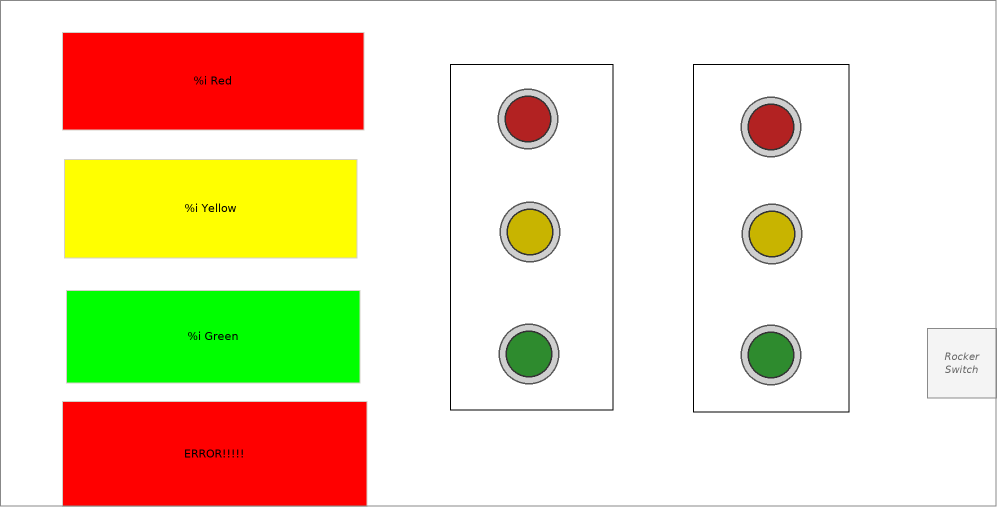
VISUALIZATION Visualization  // 997x507
    Rectangle (450,64 163x346)
    Lamp1 (494,319 70x70), variable: TrafficLight.bGreenLight, style: Lamp-Lamp1-Green
    Lamp1 (495,197 70x70), variable: TrafficLight.bYellowLight, style: Lamp-Lamp1-Yellow
    Lamp1 (493,84 70x70), variable: TrafficLight.bRedLight, style: Lamp-Lamp1-Red
    RockerSwitch (927,328 70x70), variable: TrafficLight.bTurnOnVis, behaviour: TOGGLE, style: Switch-RockerSwitch-Red
    Textfield (62,32 302x98), "%i Red", text variable: TrafficLight.iRedColor
        OnMouseDown: write the text variable via Default
    Textfield (64,159 293x99), "%i Yellow", text variable: TrafficLight.iYellowColor
        OnMouseDown: write the text variable via Default
    Textfield (62,401 305x106), "ERROR!!!!!", invisible if: NOT TrafficLight.bTextError
    Textfield (66,290 294x93), "%i Green", text variable: TrafficLight.iGreenColor
        OnMouseDown: write the text variable via Default
    Rectangle (693,64 156x348)
    Lamp1 (736,92 70x70), variable: TrafficLight.bRedLight2nd, style: Lamp-Lamp1-Red
    Lamp1 (737,199 70x70), variable: TrafficLight.bYellowLight2nd, style: Lamp-Lamp1-Yellow
    Lamp1 (736,320 70x70), variable: TrafficLight.bGreenLight2nd, style: Lamp-Lamp1-Green
END_VISUALIZATION

(* stored: Version 1.1.0.1, ProductVersion 3.1.4024.12
   Visu Visualization: Id {b6221f23-3b09-46ff-b8b7-853ddd1ae8d1} *)
